Staubli VAL3: getConvSpeed.pgx

public program getConvSpeed(num x_nConvNum (dimensions=1), num& x_nSpeed[] (dimensions=1), num& x_nError[] (dimensions=1))
begin
  // This program returns the speed of the conveyor number passed as parameter
  //
  // Input Param
  //  x_nConvNum  : Conveyor number
  //
  // Output Param
  //  x_nSpeed    : conveyor speed
  //  x_nError    : Error code
  //    0    --> No error
  //    3    --> Invalid conveyor number
  //
  //----------------------------------------------------------------
  //
  if x_nConvNum>size(nConveyorSpeed)-1
    x_nError=3
  else
    x_nError=0
    x_nSpeed=nConveyorSpeed[x_nConvNum]
  endIf
end
